FUNCTION_BLOCK Aborting_State  IMPLEMENTS ITF_State
VAR_INPUT
END_VAR
VAR_OUTPUT
END_VAR
VAR
	pPML_Base : POINTER TO PML_StatePattern_Base;
	_stateMachine : IPmlStateMachine;
END_VAR

METHOD Cycle : BOOL
_stateMachine.SetStateComplete();
pPML_Base^.SetState(pPML_Base^.aborted);
END_METHOD

METHOD FB_init : BOOL
VAR_INPUT
	bInitRetains : BOOL; // if TRUE, the retain variables are initialized (warm start / cold start)
	bInCopyCode : BOOL;  // if TRUE, the instance afterwards gets moved into the copy code (online change)
	pPML_Base : POINTER TO PML_StatePattern_Base;
	statemachine : IPmlStateMachine;
END_VAR
_stateMachine := statemachine;
THIS^.pPML_Base := pPML_Base;
END_METHOD

END_FUNCTION_BLOCK

(* stored: Version 1.1.0.1, ProductVersion 3.1.4024.12
   POU Aborting_State: Id {9ad29b47-7330-4ef2-b0c5-59754296754f}, SpecialFunc None
   Method Cycle: Id {fec74ea0-3475-4a7b-9c64-7b4a1d2a7e0a}
   Method FB_init: Id {e57274ba-de98-4eeb-b5e8-8765fcac59eb} *)
